TEXTLIST languageSupport
  axesAvailable = 'PLC Axes available: %d' | Test: 'Alt language'
  velocity = 'Velocity:'
  actposition = 'Actual Position:'
  enable = 'Enable Axis'
  enFW = 'Fwd Enable'
  enBW = 'Bwd Enable'
  axisSel = 'Axis Selected:'
  actVelocity = 'Actual Velocity:'
  errID = 'Error ID:'
  bEnabled = 'Axis Enabled'
  bCommandAborted = 'Command Aborted'
  bBusy = 'Busy'
  bDone = 'Command Done'
  bResetDone = 'Reset Complete'
  bHomed = 'Calibrated'
  bFwEnabled = 'Fwd movement enabled'
  bBwEnabled = 'Bwd movement enabled'
  bError = 'Error'
  fVelocity = 'Target Velocity:'
  fAcceleration = 'Target Accel.:'
  fDeceleration = 'Target Decel.:'
  fPosition = 'Target Position:'
  moveAbsolute = 'Absolute position move'
  toggle = 'Toggle'
  moveVelocity = 'Constant velocity move'
  bExecute = 'Motion function executed'
  moveRelative = 'Relative position move'
  moveModulo = 'Modulo position move'
  reset = 'Reset axis'
  stop = 'Stop motion'
  jogBw = 'Jog Backward'
  jogFw = 'Jog Forward'
  bGeared = 'In Gear'
  masterGear = 'Master Axis'
  gearRatio = 'Gear Ratio'
  gearIn = 'Gear In'
  gearOut = 'Gear Out'
  eHomeToLimit_Bwd = 'Bwd Limit'
  eHomeToLimit_Fwd = 'Fwd Limit'
  eHomeToRef_Bwd = 'Home Switch Bwd '
  eHomeToRef_Fwd = 'Home Switch Fwd '
  eHomeToEncPulse_Bwd = 'Enc Index Bwd '
  eHomeToEncPulse_Fwd = 'Enc Index Fwd'
  eHomeToEncPulse_viaBwdLimit = 'Enc Index via Bwd Limit'
  eHomeToEncPulse_viaFwdLimit = 'Enc Index via Fwd Limit'
  eHomeToBlock_Bwd = 'Home To Block Bwd'
  eHomeToBlock_Fwd = 'Home To Block Fwd'
  eHomeDirect = 'Home Direct'
  fHomePosition = 'Set Pos after Homing'
  fHomeFinishDistance = 'Relative Move after Homing'
  halt = 'Halt Motion'
  bInterlockBwd = 'Interlock Bwd'
  bInterlockFwd = 'Interlock Fwd'
  Home = 'HOME'
  eWriteParameter = 'Write Parameter'
  eReadParameter = 'Read Parameter'
  fWriteAxisParameter = 'Parameter to write'
  fReadAxisParameter = 'Parameter'
  bLocalMode = 'Local Mode'
  bInVelocity = 'Target velocity reached'
  bHighTempAxisDisabled = 'Disabled by High Temp '
  fActualTemp = 'Actual Temp'
  bHWMaskActive = 'HW Mask Active'
  bMoving = 'Moving'
   = ''
END_TEXTLIST

(* stored: Version 1.1.0.1, ProductVersion 3.1.4024.12
   TextList languageSupport: Id {5d3fdc2f-5bea-44d3-8108-bdef8127e821} *)
